# EPICS substitutions: iocs/visarCameraIOC/visarCameraApp/Db/visarCameraIOC.substitutions
file ADBase.template
{
	{
	P		= $(P),
	R		= $(R),
	PORT	= $(PORT),
	ADDR	= $(ADDR),
	TIMEOUT	= $(TIMEOUT)
	}
}

file visarCamera.template
{
	{
	P				= $(P),
	R				= $(R),
	PORT	= $(PORT),
    ADDR	= $(ADDR),
    TIMEOUT	= $(TIMEOUT),
    PORTC           =$(PORTC),
    PORTC2           =$(PORTC2),
    PORTD           =$(PORTD)
	}
}
